FUNCTION_BLOCK FB_CTUD_LINT (* counters (up-down-counter) *)
  (* Standard: 61131-3; Classification: counters *)
  (* Version 1.0, 2009-09-14, 4DIAC-IDE, 4DIAC-Consortium *)
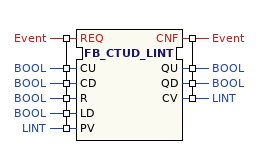
  EVENT_INPUT
    REQ WITH CD, PV, LD, CU, R; (* Service Request *)
  END_EVENT
  EVENT_OUTPUT
    CNF WITH QU, CV, QD; (* Confirmation of Requested Service *)
  END_EVENT
  VAR_INPUT
    CU : BOOL; (* Count up (Rising Edge Detection) *)
    CD : BOOL; (* Count down (Rising Edge Detection) *)
    R : BOOL; (* Reset *)
    LD : BOOL; (* Load *)
    PV : LINT; (* Preset value *)
  END_VAR
  VAR_OUTPUT
    QU : BOOL; (* Output up count *)
    QD : BOOL; (* Output down count *)
    CV : LINT; (* Count value *)
  END_VAR
  (* Service APPLICATION/RESOURCE: counters (up-down-counter) *)
END_FUNCTION_BLOCK
